Universal Robots PolyScope program: ReadSinglePosition.urp

ProgramRoot directory=/home/ur/ursim-3.1/programs/Howtos; kinematics=(a=[0, -0.425, -0.39225, 0, 0, 0], d=[0.08916, 0, 0, 0.10915, 0.09465, 0.0823], alpha=[1.5708, 0, 0, 1.5708, -1.5708, 0], deltaTheta=[0, 0, 0, 0, 0, 0], status=notInitialized); lastSavedInVersion=(project__name=Polyscope, major__version=3, minor__version=1, svn__revision=17195, build__date=Mar 11 2015, 13:02:28); name=ReadSinglePosition; programVersion=(project__name=Polyscope, major__version=3, minor__version=1, svn__revision=17195, build__date=Mar 11 2015, 13:02:28); robotEnvironmentFileName=default; serialNumberRobot=2014350001
  MainProgram cartesianAcceleration=1.2; cartesianSpeed=0.25; jointAcceleration=1.3962634015954636; jointSpeed=1.0471975511965976; sharedProcessMoveBlendRadius=0.025; motionType=JOINT_SPACE
    Move cartesianAcceleration=1.2; cartesianSpeed=0.25; jointAcceleration=1.3962634015954636; jointSpeed=1.0471975511965976; sharedProcessMoveBlendRadius=0.025; motionType=JOINT_SPACE
      Waypoint blendRadius=0.05; cartesianAcceleration=1.2; cartesianSpeed=0.25; jointAcceleration=1.3962634015954636; jointSpeed=1.0471975511965976; nextMotionTime=2.0; stoppoint=true; useSharedBlendParameter=true; useSharedParameters=true; position=TCP in base x=245.566 y=284.565 z=146.072 mm, rx=2.5949 ry=-1.7583 rz=-0.0545 rad; joints [65.626, -89.63, -137.135, -43.27, 92.027, 43.867] deg; positionType=FIXED_POSITION; waypointPoseInFeatureCoordinates=(pos=(x=0.24556557552389527, y=0.2845646077484439, z=0.14607245828364773), rot=(x=2.5949451209511434, y=-1.758288746494386, z=-0.05448385003618043)); name=Waypoint_1
    Comment commentString=Save robot position to CurrPose
    Assignment expr=get_actual_tcp_pose(); operatorValueType=INTEGER; valueSource=EXPRESSION
    Comment commentString=Save the Y parameter to Y_pos
    Assignment expr=ExpressionVariableNode[1]; operatorValueType=INTEGER; valueSource=EXPRESSION
    Comment commentString=Save the joint positions to CurrRot
    Assignment expr=get_actual_joint_positions(); operatorValueType=INTEGER; valueSource=EXPRESSION
    Comment commentString=Save rotation on Elbow to Rot_Elbow
    Assignment expr=ExpressionVariableNode[2]; operatorValueType=INTEGER; valueSource=EXPRESSION
